TYPE (* ISOBUS UT scroll list object pool properties (list + scrollbar geometry) *)
  (* Standard: 61499-2; Description: Copyright (c) 2026 Meisterschulen am Ostbahnhof This program and the accompanying materials are made available under the terms of the Eclipse Public License 2.0 which is available at https://www.eclipse.org/legal/epl-2.0/ SPDX-License-Identifier: EPL-2.0 *)
  (* Version 1.0, 2026-08-09, Franz Höpfinger, Meisterschulen am Ostbahnhof, initial API and implementation and/or initial documentation *)
  PACKAGE isobus::utils::scroll;
  IMPORT isobus::UT::Q::const::IDs;
  ScrollObjectPool_S : STRUCT
    u16ListParentId : UINT := IDs::ID_NULL; (* Object ID of the list viewport container (Change Child Position parent) *)
    u16ListContentId : UINT := IDs::ID_NULL; (* Object ID of the moved list content container (Change Child Position child) *)
    i32RowHeight : DINT := 0; (* Row height in pixels *)
    u16BarParentId : UINT := IDs::ID_NULL; (* Object ID of the scrollbar viewport container (Change Child Position parent) *)
    u16BarContentId : UINT := IDs::ID_NULL; (* Object ID of the moved scrollbar indicator content container (Change Child Position child) *)
    i32BarBaseOffset : DINT := 0; (* BarContent.Top at position 0 (negative of the indicator's fixed internal Top) *)
    i32BarTravel : DINT := 0; (* Total pixels the indicator travels: window height minus indicator height *)
    i32PosMax : DINT := 0; (* Upper bound of the scroll position: row count minus visible rows *)
    i32Step : DINT := 1; (* Step size for the fast (page) scroll events *)
  END_STRUCT;
END_TYPE
